(* PLC project Unnamed, Unknown Unnamed 1 *)
(* stored: creationDateTime 2019-08-06T14:23:42, modificationDateTime 2020-09-23T16:29:40 *)

FUNCTION_BLOCK PumpControl
  VAR
    Pump : HMI_NODE;
    Pressure : HMI_INT;
  END_VAR
  VAR_INPUT
    TargetPressure : INT;
  END_VAR
  VAR
    Sloth : HMI_INT;
    boolout : HMI_BOOL;
    boolin : HMI_BOOL := True;
    strout : HMI_STRING;
    strin : HMI_STRING := blup;
  END_VAR
  VAR  (* added by the conversion: wires and edge detectors of the diagram *)
    _ADD6_OUT : INT;
  END_VAR

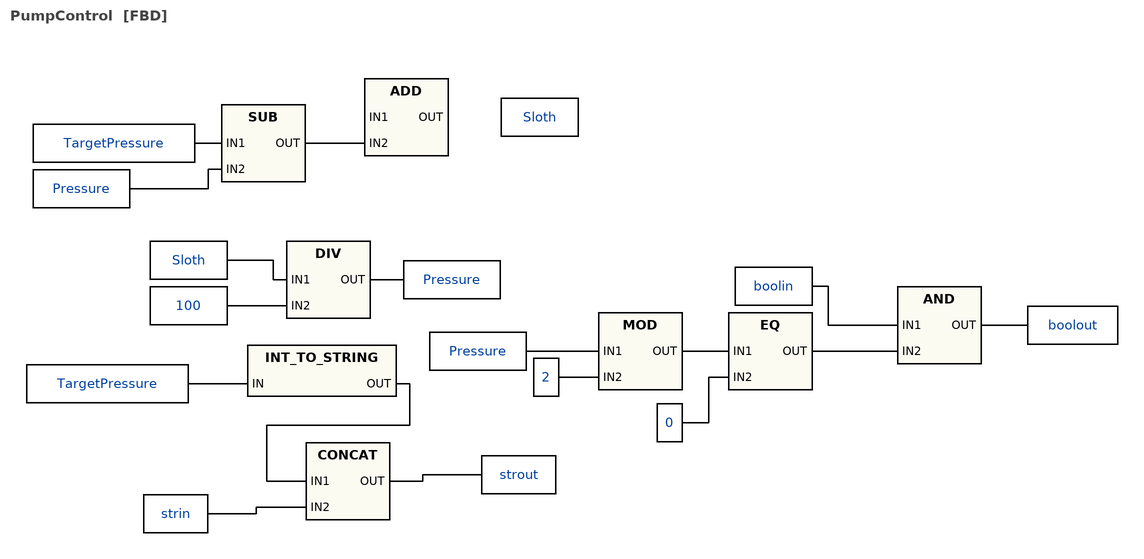
(* FBD diagram, written out as Structured Text *)
Pressure := Sloth / 100;
boolout := boolin AND Pressure MOD 2 = 0;
strout := CONCAT(INT_TO_STRING(TargetPressure), strin);
_ADD6_OUT := ADD(IN2 := TargetPressure - Pressure);
(* drawn but not wired to any output: Sloth *)
END_FUNCTION_BLOCK

PROGRAM MainStuff
  VAR
    TargetPressure : HMI_INT;
    selection : HMI_INT;
    Pump0 : PumpControl;
    TestButton : HMI_BOOL;
    TestLocal : BOOL;
    Multistate : HMI_INT;
    Radiostate : HMI_INT;
    Toggle : HMI_BOOL;
    Toggle1 : HMI_BOOL;
    Toggle2 : HMI_BOOL;
    MultistateExt : INT;
    Speed : HMI_REAL;
  END_VAR

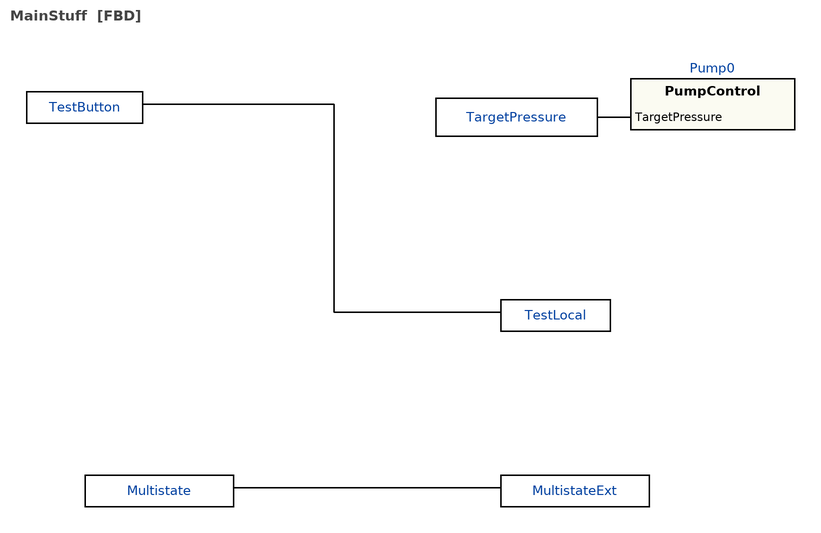
(* FBD diagram, written out as Structured Text *)
TestLocal := TestButton;
MultistateExt := Multistate;
Pump0(TargetPressure := TargetPressure);
END_PROGRAM

CONFIGURATION config
  RESOURCE resource1 ON PLC
    TASK task0(INTERVAL := T#20ms, PRIORITY := 0);
    PROGRAM instance0 WITH task0 : MainStuff;
  END_RESOURCE
END_CONFIGURATION
